// Brief: Slave Arm joint3 retract to up limit
FUNCTION_BLOCK PUBLIC FB_SlaveCtrlInstruRetract EXTENDS FB_SlaveArmCtrlBase
VAR_INPUT
END_VAR
VAR_OUTPUT
END_VAR
VAR
	// wait time before retract, ensure instruments is removed 
	m_waitTime :LREAL :=2.0;
		
	// motion planning
	m_jnt3OTG : FB_secOrdTrajFilter;
	m_jnt3TargetPos :LREAL;
	m_retractVel: LREAL:= 0.1;
	m_retractAcc: LREAL:= 0.2;
	
	// instrument joint motion planning
	m_instruJntOTG :ARRAY[1..5] OF FB_secOrdTrajFilter;
	m_instruJntTargetPos :Vec5d;
	m_instruJntVel :LREAL := 2*PI;
	m_instruJntAcc : LREAL := 4*PI;
	
	// PID for joint8
//	m_retractCtrl : FB_PID;
//	m_retractKp:LREAL:=2000;
//	m_retractKd:LREAL:=100;
//	m_retractKi:LREAL:=8000;
//	m_retractKiLimit:LREAL:=300;
//	m_retractCtrlLimit:LREAL:=1000;
	
	
END_VAR

// override this function in each exact controller
METHOD PROTECTED calcCmdJntPos : BOOL
VAR_IN_OUT CONSTANT
	i_endoscopePose : ST_Frame;
	i_masterStatus :ST_MasterStatus;
	i_setupStatus: ST_SetupStatus;
	i_slaveArm :FB_SlaveArm;
END_VAR

VAR 
	i :INT;
	trackErr:LREAL;
	curJntVel:Vec8d;
END_VAR
// if instrument is on again, wait and re-plan the traj
IF i_slaveArm.instruNear THEN
	m_cmdJntVel:=g_zeroVec8d;
	m_cmdJntAcc := g_zeroVec8d;
	
	// init traj filter
	m_jnt3OTG.init(m_cmdJntPos[3], 0, m_retractVel, m_retractAcc, g_slaveArmCtrlCycleTime);
	FOR i:=1 TO 5 DO
		m_instruJntOTG[i].init(m_cmdJntPos[i+3], 0,m_instruJntVel, m_instruJntAcc, g_slaveArmCtrlCycleTime);
	END_FOR

	m_timePeriod := 0;
	RETURN;
END_IF

// wait
IF m_timePeriod< m_waitTime THEN
	RETURN;
END_IF

// traj plan
m_jnt3OTG.run(m_jnt3TargetPos, 0.0, o_cmdAcc=>m_cmdJntAcc[3],o_cmdVel=>m_cmdJntVel[3],o_cmdPos=>m_cmdJntPos[3]);
FOR i:=1 TO 5 DO
	m_instruJntOTG[i].run(m_instruJntTargetPos[i], 0.0, o_cmdAcc=>m_cmdJntAcc[i+3],o_cmdVel=>m_cmdJntVel[i+3],o_cmdPos=>m_cmdJntPos[i+3]);
END_FOR

// reach target check
trackErr :=0;
FOR i:=1 TO 5 DO 
	trackErr := MAX(trackErr, ABS(m_cmdJntPos[i+3]-m_instruJntTargetPos[i]));
END_FOR
curJntVel := i_slaveArm.curJntVel;
m_isFinished := (ABS(m_cmdJntPos[3] - m_jnt3TargetPos) <g_cartCtrlPosTolLow AND trackErr < g_jntCtrlAngTolLoW 
			AND norm(curJntVel) <g_jntStaticVelThres);
END_METHOD

// override this function in each exact controller
METHOD PROTECTED calcCmdJntTrq : BOOL
VAR_IN_OUT CONSTANT
	i_endoscopePose : ST_Frame;
	i_masterStatus :ST_MasterStatus;
	i_setupStatus: ST_SetupStatus;
	i_slaveArm :FB_SlaveArm;
END_VAR
VAR
	i :INT;
	dampScale :LREAL;
	limitDis:LREAL;
END_VAR
// TODO: re-tune joint3 controller, replace this local PID controller with the global one if possible
m_cmdJntTrq := g_zeroVec8d;
END_METHOD

METHOD PUBLIC init : BOOL
VAR_IN_OUT CONSTANT
	i_slaveArm	:FB_SlaveArm;
END_VAR
VAR_IN_OUT 
	r_slaveArmCtrlCmd :ST_SlaveArmCtrlCmds;
END_VAR

VAR
	i:INT;
	cycleNum:LREAL;
END_VAR
// check if to hold the command joint position unchanged
m_holdLastCmds := checkToHoldLastCmds(i_slaveArm);

SUPER^.Init(i_slaveArm,r_slaveArmCtrlCmd);

// decide target position
m_jnt3TargetPos := GVL_SlaveMotorParameters.g_maxDHJntPos[3]-i_slaveArm.m_caliJntPosErr[3];

// init traj filter
m_jnt3OTG.init(m_cmdJntPos[3], 0, m_retractVel, m_retractAcc, g_slaveArmCtrlCycleTime);

// set wait time before start retract
IF SlaveArmControl.m_slaveRobot.m_lastSlaveArmState[i_slaveArm.armIdx] = SlaveArmState_PanelReady THEN
	m_waitTime := 0;
ELSE
	m_waitTime :=1.0;
END_IF

// decide instrument joint zero position and init traj filter
FOR i:=1 TO 5 DO
	cycleNum := FLOOR(i_slaveArm.curJntPos[i+3]/g_2pi);
	m_instruJntTargetPos[i]:=cycleNum* g_2Pi;
	m_instruJntOTG[i].init(m_cmdJntPos[i+3], 0,m_instruJntVel, m_instruJntAcc, g_slaveArmCtrlCycleTime);
END_FOR

// update commands to arm
copyCmds(r_slaveArmCtrlCmd);
END_METHOD

END_FUNCTION_BLOCK

(* stored: Version 1.1.0.1, ProductVersion 3.1.4024.11
   POU FB_SlaveCtrlInstruRetract: Id {596332da-68eb-4244-8a80-7e3d57b3bb9f}, SpecialFunc None
   Method calcCmdJntPos: Id {7b11d094-8bfe-4cb8-971c-9702c727740e}
   Method calcCmdJntTrq: Id {24cd49e3-93cf-41f3-8feb-c2dc5ff73b79}
   Method init: Id {7aae2cb5-3dc8-47a4-84c8-fce1eb91d921} *)
